TYPE "ST_SpkCylinderOutImm"
VERSION : 0.1
   STRUCT
      Extended : Bool;
      Retracted : Bool;
   END_STRUCT;

END_TYPE
